{attribute 'qualified_only'}
{attribute 'strict'}
TYPE Camera_Type :
(
	Cognex_7000 := 0,
	Cognex_5100 := 1
)UINT;
END_TYPE

(* stored: Version 1.1.0.1, ProductVersion 3.1.4024.10
   DUT Camera_Type: Id {95fa2ca1-80d1-4984-ba1e-eee1c90130d8} *)
